PROGRAM MAIN
VAR
	Servo : StructAxis;		//CONV 1
	Stepper : StructAxis;	//CONV2
	
	ServoAxis : AXIS_REF;
	StepperAxis : AXIS_REF;
	oState : Conv2;
	iState : Conv1;
	
	tim1 : TON;
END_VAR

ACT_Move();
ACT_Power();
ACT_Reset();
ACT_Stop();

CASE iState OF 
	Conv1.Init: 						// setting intial position of Conv1
		tim1(IN:=FALSE);
		servo.MoveVel.Execute :=FALSE;  
		servo.Reset.Execute :=FALSE;
		
		iState := Conv1.Enable; // move to next step(enabling servo motor)
		
	Conv1.Enable:					// Power up the Servo motor
		servo.Power.Enable := TRUE;
		servo.Power.Enable_Positive := TRUE;
	    servo.Power.Enable_Negative := TRUE;
		
		IF servo.Power.Status THEN
			iState := Conv1.Conv1ON;
 		ELSIF servo.Power.Error THEN
			iState := Conv1.Error;
		END_IF
		
	Conv1.Conv1ON:
		IF IO.bSwitch1 THEN						// Start button pressed
			IO.bLed1 := TRUE;					// show logic works
			iState := Conv1.MoveForwards;// Conv1 move forward
		
		END_IF
	Conv1.MoveForwards:
		tim1(IN:=FALSE);
	
		Servo.MoveVel.Execute := TRUE;
		Servo.MoveVel.Velocity := 100;
	
		IF IO.bSwitch2 THEN					// if "Box" is detected on Conv1
			IO.bLed2 := TRUE;
			servo.MoveVel.Execute := FALSE;
			iState := Conv1.Conv1Stop; 		// Conv1 Stop
		IF IO.bSwitch2 AND IO.bSwitch4 THEN
			iState := Conv1.tim1;
		END_IF
		END_IF
		
	Conv1.tim1:
			tim1(IN := TRUE,PT := T#5S);
			IF tim1.Q THEN
				iState := Conv1.MoveForwards;
			END_IF
			
	Conv1.Conv1Stop:
		Servo.McStop.Execute := TRUE;
				
		IF Servo.McStop.Done THEN
			Servo.McStop.Execute := FALSE;
			iState := Conv1.MoveForwards;
		END_IF
		
	IF servo.MoveVel.Error OR servo.MoveVel.CommandAborted THEN // if error or sudden estop initiated
			iState := Conv1.Error;
			stepper.MoveVel.Execute :=FALSE;
			
		END_IF
		
	Conv1.Error:													// if error, stop n reset
		IF StepperAxis.Status.Error  THEN
			iState := Conv1.Reset;
		ELSE
			iState := Conv1.Init;
		END_IF
		
	Conv1.Reset:
		Servo.Reset.Execute := TRUE;
		
		
		IF  servo.Reset.Done THEN
			iState := Conv1.Init;
		ELSIF servo.Reset.Error THEN
			iState := Conv1.Error;
		END_IF
	
	

END_CASE
//////////////////////////////////////////////////////////////////////////////////////////////////////////////////////////////////////////////////////////////////////////////////////////////////////////////
			CASE oState OF 
				Conv2.Init: 						// setting intial position of Conv2
					Stepper.MoveVel.Execute :=FALSE;  
					stepper.Reset.Execute :=FALSE;
					Servo.McStop.Execute := FALSE;
					oState := Conv2.Enable; // move to next step(enabling stepper motor)
					
				Conv2.Enable:					// Power up the stepper motor
					stepper.Power.Enable := TRUE; 
					stepper.Power.Enable_Positive := TRUE; // Ensure it is able to turn positive and negative
					stepper.Power.Enable_Negative := TRUE;
				   
					
					IF Stepper.Power.Status THEN
						oState := Conv2.Conv2ON;
			 		ELSIF Stepper.Power.Error THEN
						oState := Conv2.Error;
					END_IF
					
				Conv2.Conv2ON:
					IF IO.bSwitch1 THEN						// Start button pressed
						IO.bLed1 := TRUE;					// show logic works
						oState := Conv2.MoveForwards;		// Conv2 move forward
					ELSE IO.bLed1 := FALSE;
					END_IF
					
				Conv2.MoveForwards:
				
						stepper.MoveVel.Execute := TRUE;
						stepper.MoveVel.Velocity := 100;
					
					IF IO.bSwitch3 THEN					// if "Object" is detected on Conv2
						IO.bLed3 := TRUE;
						Stepper.MoveVel.Execute := FALSE;
						oState := Conv2.Conv2Stop;	 	// Conv2 Stop
					END_IF
					
				Conv2.Conv2Stop:
					stepper.McStop.Execute := TRUE;
							
					IF NOT IO.bSwitch3 THEN
						Stepper.McStop.Execute := FALSE;
						oState := Conv2.MoveForwards;
					END_IF
					
				IF Stepper.MoveVel.Error OR Stepper.MoveVel.CommandAborted THEN // if error or sudden estop initiated
						oState := Conv2.Error;
						stepper.MoveVel.Execute :=FALSE;
						
					END_IF
					
				Conv2.Error:													// if error, stop n reset
					IF StepperAxis.Status.Error  THEN
						oState := Conv2.Reset;
					ELSE
						oState := Conv2.Init;
					END_IF
					
				Conv2.Reset:
					Stepper.Reset.Execute := TRUE;
					
					IF  Stepper.Reset.Done THEN
						oState := Conv2.Init;
					ELSIF Stepper.Reset.Error THEN
						oState := Conv2.Error;
					END_IF
				
			END_CASE

ACTION ACT_Move:
Servo.MoveVel(Axis := ServoAxis);
	
Stepper.MoveVel( Axis := StepperAxis);
END_ACTION

ACTION ACT_Power:
Servo.Power( Axis := ServoAxis);

Stepper.Power( Axis := StepperAxis);
END_ACTION

ACTION ACT_Reset:
Servo.Reset( Axis := ServoAxis);

Stepper.Reset( Axis := StepperAxis);
END_ACTION

ACTION ACT_Stop:
Servo.McStop(Axis := ServoAxis);
	
Stepper.McStop( Axis := StepperAxis);
END_ACTION

END_PROGRAM

(* stored: Version 1.1.0.1, ProductVersion 3.1.4024.10
   POU MAIN: Id {07b3dce6-b628-40b9-a967-2b66a8008996}, SpecialFunc None
   Action ACT_Move: Id {176658c8-fa86-43f2-9e39-a51b8813feed}
   Action ACT_Power: Id {d7d186e7-98bf-409e-9dd7-518f5e3b9bd6}
   Action ACT_Reset: Id {0ed80840-1307-4a41-af3f-cbaf470eb74d}
   Action ACT_Stop: Id {da3ba7eb-524f-477c-8948-77cf9c74676d} *)
